(* Logix 5000 project; controller Sucrose_Main Emulate 5570 rev 20.12; software revision 20.01; part 18 of 30 *)
(* tags used below, declared in another part *)
   Alarm_ACK_Master_Timer : TIMER;
   DO_E22_6 : ALIAS FOR FLX_E22:6:O;   // Discrete Output EN2T_FLX 192.168.1.22
   DO_E22_7 : ALIAS FOR FLX_E22:7:O;   // Discrete Output EN2T_FLX 192.168.1.22
   FV740401_AOI : QSI_Flow_Valve;   // FV-74-04-01 SIP SUPPLY VALVE
   FV740501_AOI : QSI_Flow_Valve;   // FV-74-05-01 SIP SUPPLY TO PRE FILTER TRAIN 1 VALVE
   FV740502_AOI : QSI_Flow_Valve;   // FV-74-05-02 SIP SUPPLY TO FINAL FILTER TRAIN 1 VALVE
   FV740601_AOI : QSI_Flow_Valve;   // FV-74-06-01 SIP SUPPLY TO PRE FILTER TRAIN 2 VALVE
   FV740602_AOI : QSI_Flow_Valve;   // FV-74-06-02 SIP SUPPLY TO FINAL FILTER TRAIN 2 VALVE
   FV750501_AOI : QSI_Flow_Valve;   // FV-75-05-01 TRP-75-05-01 ISOLATION VALVE
   FV750502_AOI : QSI_Flow_Valve;   // FV-75-05-02 TRP-75-05-02 ISOLATION VALVE
   FV750503_AOI : QSI_Flow_Valve;   // FV-75-05-03 TRP-75-05-03 ISOLATION VALVE
   FV750504_AOI : QSI_Flow_Valve;   // FV-75-05-04 TRP-75-05-04 ISOLATION VALVE
   FV750601_AOI : QSI_Flow_Valve;   // FV-75-06-01 TRP-75-06-01 ISOLATION VALVE
   FV750602_AOI : QSI_Flow_Valve;   // FV-75-06-02 TRP-75-06-02 ISOLATION VALVE
   FV750603_AOI : QSI_Flow_Valve;   // FV-75-06-03 TRP-75-06-03 ISOLATION VALVE
   FV750604_AOI : QSI_Flow_Valve;   // FV-75-06-04 TRP-75-06-04 ISOLATION VALVE
   FV920501_AOI : QSI_Flow_Valve;   // FV-92-05-01 FLT-23-05-01 VENT VALVE
   FV930511_AOI : QSI_Flow_Valve;   // FV-93-05-11 PRE FILTER TRAIN 1 AIR BLOW OUTLET
   FV930512_AOI : QSI_Flow_Valve;   // FV-93-05-12 FINAL FILTER TRAIN 1 AIR BLOW OUTLET
   Sucrose_MM_Enable : BOOL;
   SucroseCIP_FILTRATION_REMOTE : CIP_REMOTE;
   SucroseFiltration : Area_Program;

PROGRAM FiltrationArea_EN2T_IO_Discrete_DO_E22_6   (* main routine MainRoutine *)

ROUTINE _00_FV740401   (* ladder *)
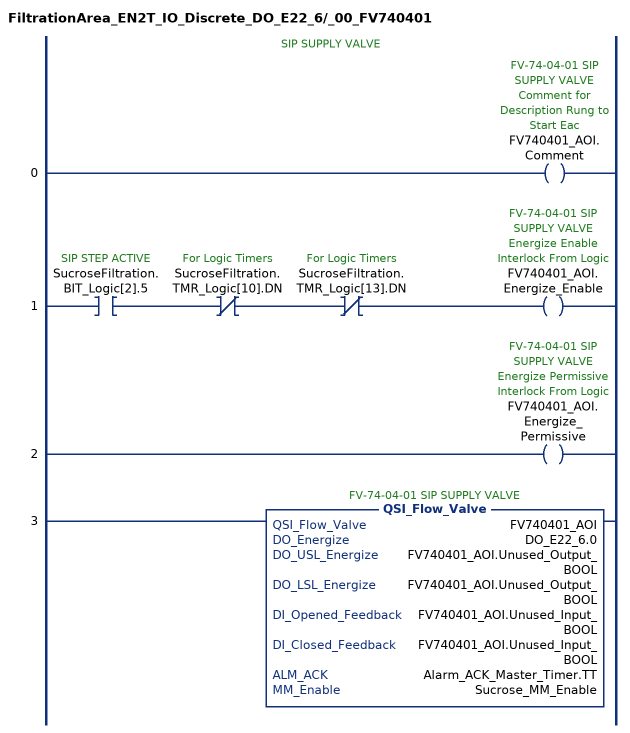
   // SIP SUPPLY VALVE
   0: OTE(FV740401_AOI.Comment);
   1: XIC(SucroseFiltration.BIT_Logic[2].5)XIO(SucroseFiltration.TMR_Logic[10].DN)XIO(SucroseFiltration.TMR_Logic[13].DN)OTE(FV740401_AOI.Energize_Enable);
   2: OTE(FV740401_AOI.Energize_Permissive);
   3: QSI_Flow_Valve(FV740401_AOI,DO_E22_6.0,FV740401_AOI.Unused_Output_BOOL,FV740401_AOI.Unused_Output_BOOL,FV740401_AOI.Unused_Input_BOOL,FV740401_AOI.Unused_Input_BOOL,Alarm_ACK_Master_Timer.TT,Sucrose_MM_Enable);
END_ROUTINE

ROUTINE _01_FV740501   (* ladder *)
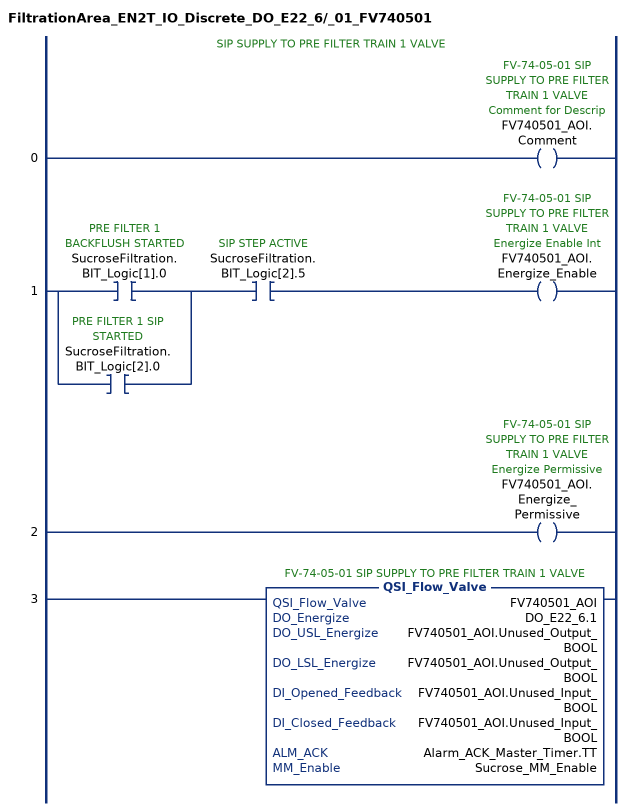
   // SIP SUPPLY TO PRE FILTER TRAIN 1 VALVE
   0: OTE(FV740501_AOI.Comment);
   1: [XIC(SucroseFiltration.BIT_Logic[1].0) ,XIC(SucroseFiltration.BIT_Logic[2].0) ]XIC(SucroseFiltration.BIT_Logic[2].5)OTE(FV740501_AOI.Energize_Enable);
   2: OTE(FV740501_AOI.Energize_Permissive);
   3: QSI_Flow_Valve(FV740501_AOI,DO_E22_6.1,FV740501_AOI.Unused_Output_BOOL,FV740501_AOI.Unused_Output_BOOL,FV740501_AOI.Unused_Input_BOOL,FV740501_AOI.Unused_Input_BOOL,Alarm_ACK_Master_Timer.TT,Sucrose_MM_Enable);
END_ROUTINE

ROUTINE _02_FV740502   (* ladder *)
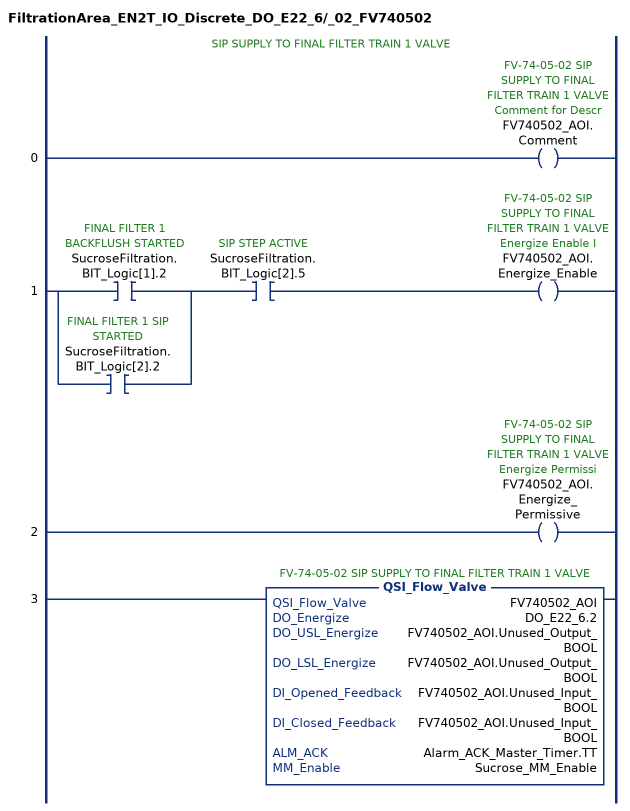
   // SIP SUPPLY TO FINAL FILTER TRAIN 1 VALVE
   0: OTE(FV740502_AOI.Comment);
   1: [XIC(SucroseFiltration.BIT_Logic[1].2) ,XIC(SucroseFiltration.BIT_Logic[2].2) ]XIC(SucroseFiltration.BIT_Logic[2].5)OTE(FV740502_AOI.Energize_Enable);
   2: OTE(FV740502_AOI.Energize_Permissive);
   3: QSI_Flow_Valve(FV740502_AOI,DO_E22_6.2,FV740502_AOI.Unused_Output_BOOL,FV740502_AOI.Unused_Output_BOOL,FV740502_AOI.Unused_Input_BOOL,FV740502_AOI.Unused_Input_BOOL,Alarm_ACK_Master_Timer.TT,Sucrose_MM_Enable);
END_ROUTINE

ROUTINE _03_FV740601   (* ladder *)
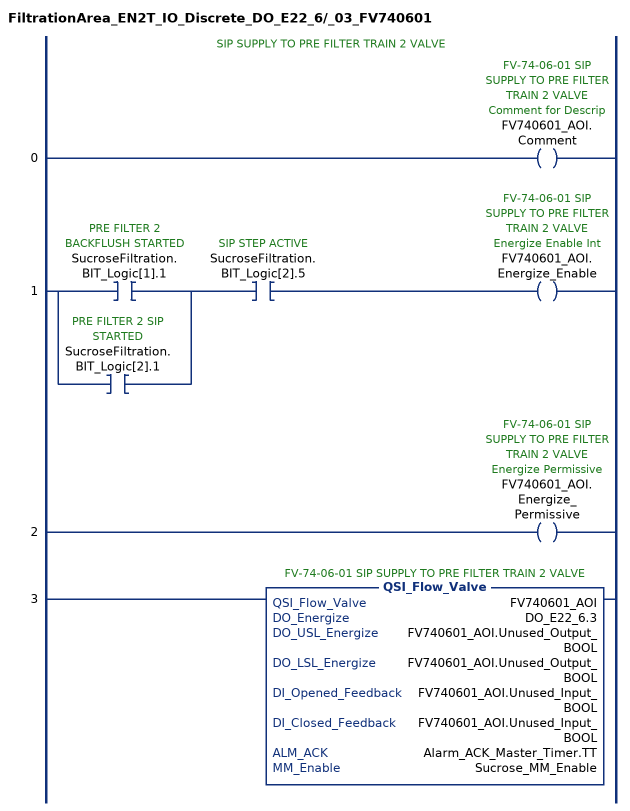
   // SIP SUPPLY TO PRE FILTER TRAIN 2 VALVE
   0: OTE(FV740601_AOI.Comment);
   1: [XIC(SucroseFiltration.BIT_Logic[1].1) ,XIC(SucroseFiltration.BIT_Logic[2].1) ]XIC(SucroseFiltration.BIT_Logic[2].5)OTE(FV740601_AOI.Energize_Enable);
   2: OTE(FV740601_AOI.Energize_Permissive);
   3: QSI_Flow_Valve(FV740601_AOI,DO_E22_6.3,FV740601_AOI.Unused_Output_BOOL,FV740601_AOI.Unused_Output_BOOL,FV740601_AOI.Unused_Input_BOOL,FV740601_AOI.Unused_Input_BOOL,Alarm_ACK_Master_Timer.TT,Sucrose_MM_Enable);
END_ROUTINE

ROUTINE _04_FV740602   (* ladder *)
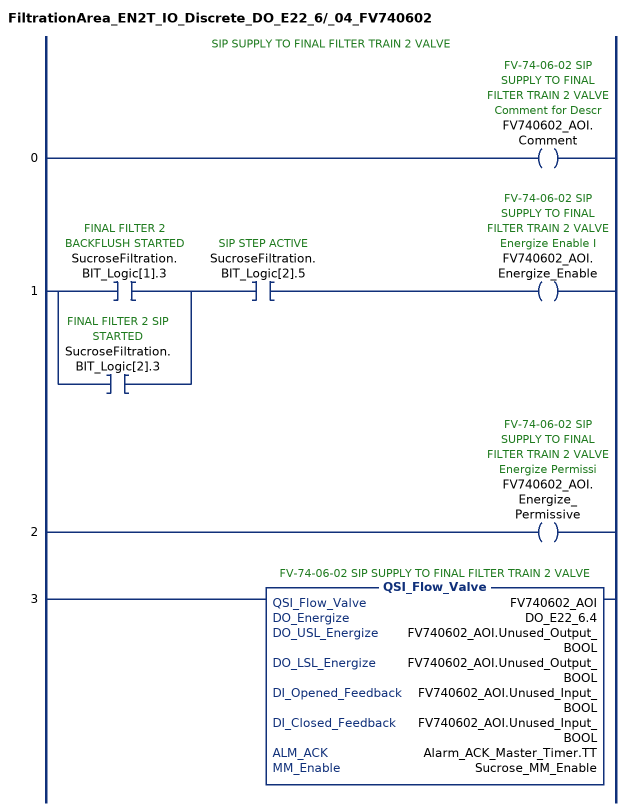
   // SIP SUPPLY TO FINAL FILTER TRAIN 2 VALVE
   0: OTE(FV740602_AOI.Comment);
   1: [XIC(SucroseFiltration.BIT_Logic[1].3) ,XIC(SucroseFiltration.BIT_Logic[2].3) ]XIC(SucroseFiltration.BIT_Logic[2].5)OTE(FV740602_AOI.Energize_Enable);
   2: OTE(FV740602_AOI.Energize_Permissive);
   3: QSI_Flow_Valve(FV740602_AOI,DO_E22_6.4,FV740602_AOI.Unused_Output_BOOL,FV740602_AOI.Unused_Output_BOOL,FV740602_AOI.Unused_Input_BOOL,FV740602_AOI.Unused_Input_BOOL,Alarm_ACK_Master_Timer.TT,Sucrose_MM_Enable);
END_ROUTINE

ROUTINE _05_FV750501   (* ladder *)
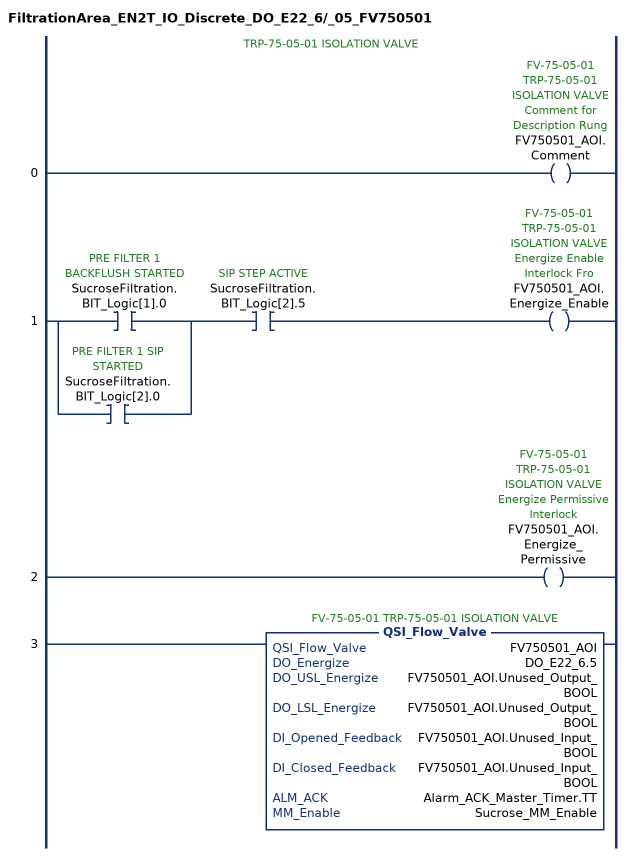
   // TRP-75-05-01 ISOLATION VALVE
   0: OTE(FV750501_AOI.Comment);
   1: [XIC(SucroseFiltration.BIT_Logic[1].0) ,XIC(SucroseFiltration.BIT_Logic[2].0) ]XIC(SucroseFiltration.BIT_Logic[2].5)OTE(FV750501_AOI.Energize_Enable);
   2: OTE(FV750501_AOI.Energize_Permissive);
   3: QSI_Flow_Valve(FV750501_AOI,DO_E22_6.5,FV750501_AOI.Unused_Output_BOOL,FV750501_AOI.Unused_Output_BOOL,FV750501_AOI.Unused_Input_BOOL,FV750501_AOI.Unused_Input_BOOL,Alarm_ACK_Master_Timer.TT,Sucrose_MM_Enable);
END_ROUTINE

ROUTINE _06_FV750502   (* ladder *)
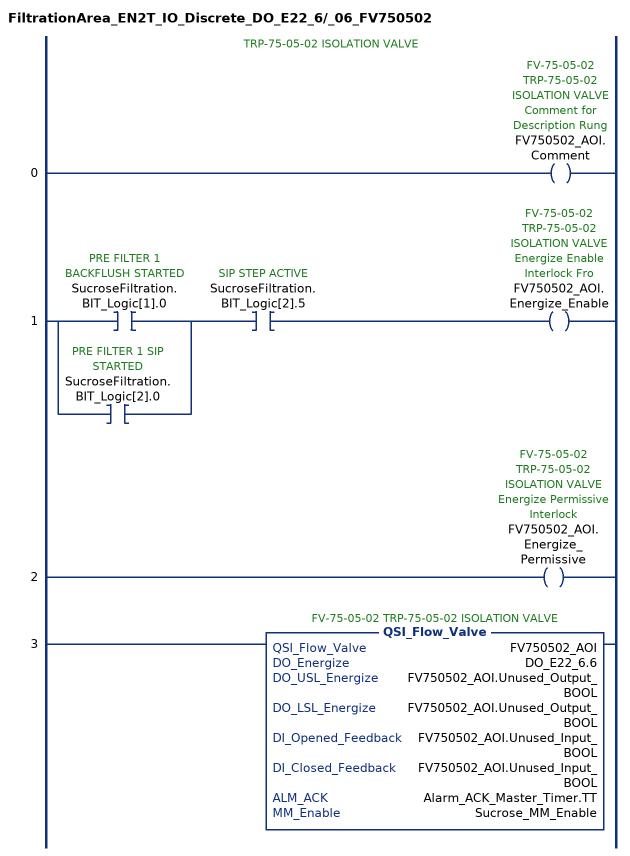
   // TRP-75-05-02 ISOLATION VALVE
   0: OTE(FV750502_AOI.Comment);
   1: [XIC(SucroseFiltration.BIT_Logic[1].0) ,XIC(SucroseFiltration.BIT_Logic[2].0) ]XIC(SucroseFiltration.BIT_Logic[2].5)OTE(FV750502_AOI.Energize_Enable);
   2: OTE(FV750502_AOI.Energize_Permissive);
   3: QSI_Flow_Valve(FV750502_AOI,DO_E22_6.6,FV750502_AOI.Unused_Output_BOOL,FV750502_AOI.Unused_Output_BOOL,FV750502_AOI.Unused_Input_BOOL,FV750502_AOI.Unused_Input_BOOL,Alarm_ACK_Master_Timer.TT,Sucrose_MM_Enable);
END_ROUTINE

ROUTINE _07_FV750503   (* ladder *)
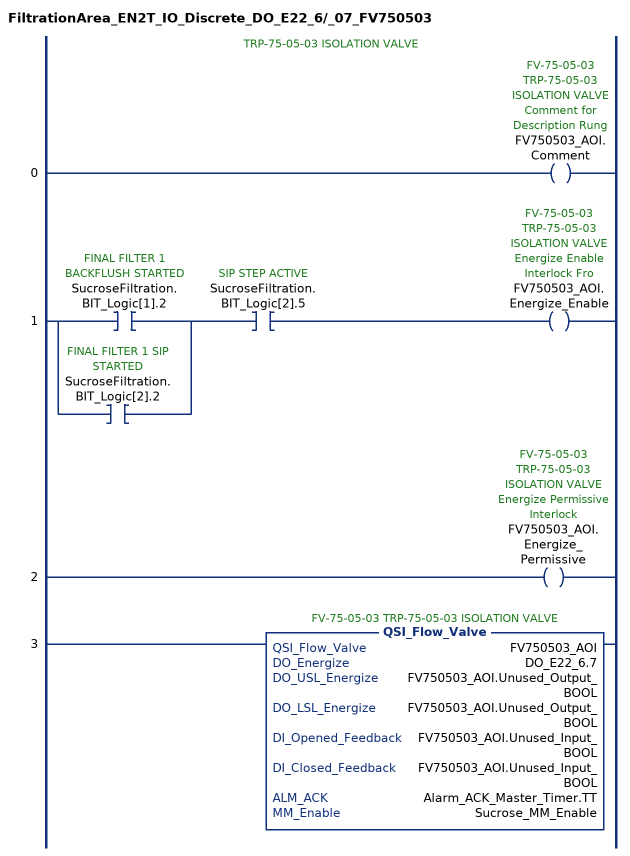
   // TRP-75-05-03 ISOLATION VALVE
   0: OTE(FV750503_AOI.Comment);
   1: [XIC(SucroseFiltration.BIT_Logic[1].2) ,XIC(SucroseFiltration.BIT_Logic[2].2) ]XIC(SucroseFiltration.BIT_Logic[2].5)OTE(FV750503_AOI.Energize_Enable);
   2: OTE(FV750503_AOI.Energize_Permissive);
   3: QSI_Flow_Valve(FV750503_AOI,DO_E22_6.7,FV750503_AOI.Unused_Output_BOOL,FV750503_AOI.Unused_Output_BOOL,FV750503_AOI.Unused_Input_BOOL,FV750503_AOI.Unused_Input_BOOL,Alarm_ACK_Master_Timer.TT,Sucrose_MM_Enable);
END_ROUTINE

ROUTINE _08_FV750504   (* ladder *)
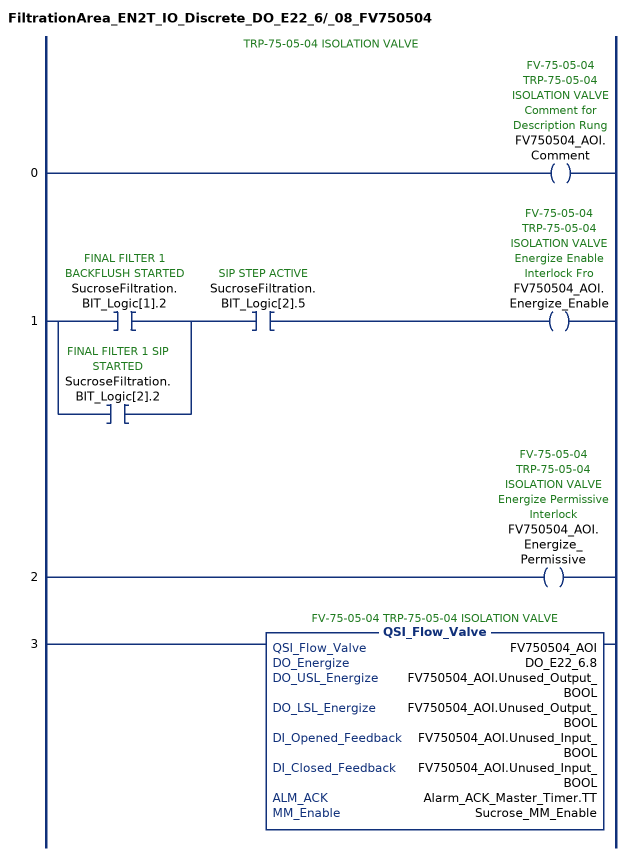
   // TRP-75-05-04 ISOLATION VALVE
   0: OTE(FV750504_AOI.Comment);
   1: [XIC(SucroseFiltration.BIT_Logic[1].2) ,XIC(SucroseFiltration.BIT_Logic[2].2) ]XIC(SucroseFiltration.BIT_Logic[2].5)OTE(FV750504_AOI.Energize_Enable);
   2: OTE(FV750504_AOI.Energize_Permissive);
   3: QSI_Flow_Valve(FV750504_AOI,DO_E22_6.8,FV750504_AOI.Unused_Output_BOOL,FV750504_AOI.Unused_Output_BOOL,FV750504_AOI.Unused_Input_BOOL,FV750504_AOI.Unused_Input_BOOL,Alarm_ACK_Master_Timer.TT,Sucrose_MM_Enable);
END_ROUTINE

ROUTINE _09_FV750601   (* ladder *)
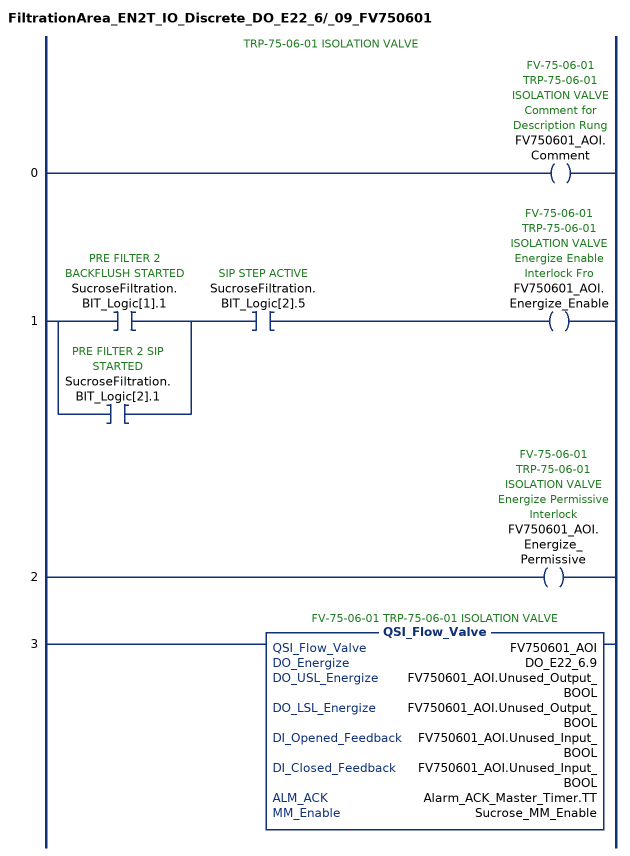
   // TRP-75-06-01 ISOLATION VALVE
   0: OTE(FV750601_AOI.Comment);
   1: [XIC(SucroseFiltration.BIT_Logic[1].1) ,XIC(SucroseFiltration.BIT_Logic[2].1) ]XIC(SucroseFiltration.BIT_Logic[2].5)OTE(FV750601_AOI.Energize_Enable);
   2: OTE(FV750601_AOI.Energize_Permissive);
   3: QSI_Flow_Valve(FV750601_AOI,DO_E22_6.9,FV750601_AOI.Unused_Output_BOOL,FV750601_AOI.Unused_Output_BOOL,FV750601_AOI.Unused_Input_BOOL,FV750601_AOI.Unused_Input_BOOL,Alarm_ACK_Master_Timer.TT,Sucrose_MM_Enable);
END_ROUTINE

ROUTINE _10_FV750602   (* ladder *)
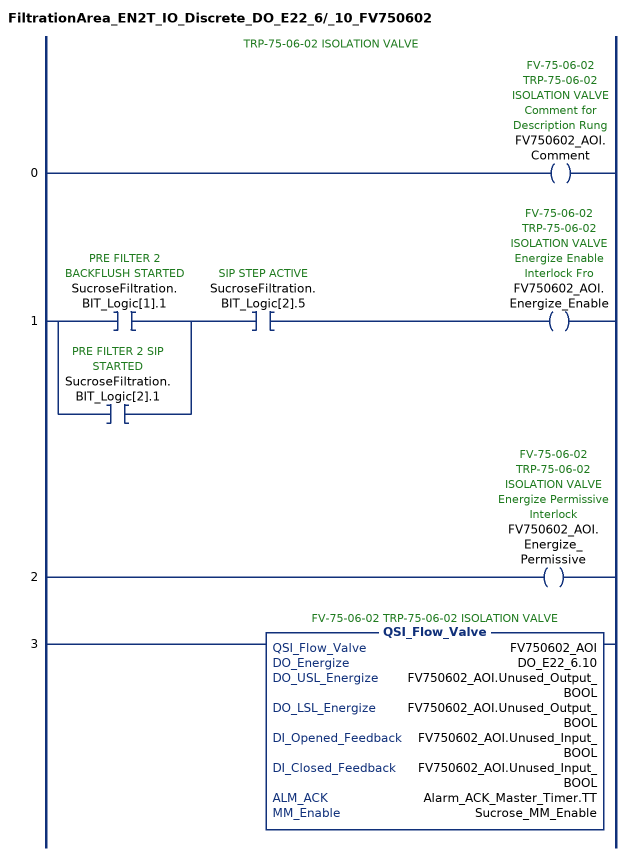
   // TRP-75-06-02 ISOLATION VALVE
   0: OTE(FV750602_AOI.Comment);
   1: [XIC(SucroseFiltration.BIT_Logic[1].1) ,XIC(SucroseFiltration.BIT_Logic[2].1) ]XIC(SucroseFiltration.BIT_Logic[2].5)OTE(FV750602_AOI.Energize_Enable);
   2: OTE(FV750602_AOI.Energize_Permissive);
   3: QSI_Flow_Valve(FV750602_AOI,DO_E22_6.10,FV750602_AOI.Unused_Output_BOOL,FV750602_AOI.Unused_Output_BOOL,FV750602_AOI.Unused_Input_BOOL,FV750602_AOI.Unused_Input_BOOL,Alarm_ACK_Master_Timer.TT,Sucrose_MM_Enable);
END_ROUTINE

ROUTINE _11_FV750603   (* ladder *)
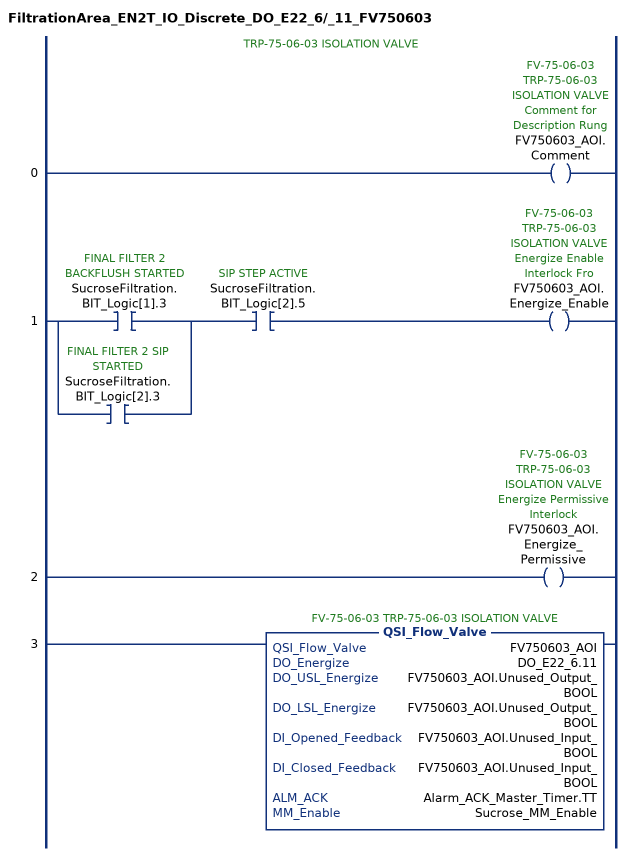
   // TRP-75-06-03 ISOLATION VALVE
   0: OTE(FV750603_AOI.Comment);
   1: [XIC(SucroseFiltration.BIT_Logic[1].3) ,XIC(SucroseFiltration.BIT_Logic[2].3) ]XIC(SucroseFiltration.BIT_Logic[2].5)OTE(FV750603_AOI.Energize_Enable);
   2: OTE(FV750603_AOI.Energize_Permissive);
   3: QSI_Flow_Valve(FV750603_AOI,DO_E22_6.11,FV750603_AOI.Unused_Output_BOOL,FV750603_AOI.Unused_Output_BOOL,FV750603_AOI.Unused_Input_BOOL,FV750603_AOI.Unused_Input_BOOL,Alarm_ACK_Master_Timer.TT,Sucrose_MM_Enable);
END_ROUTINE

ROUTINE _12_FV930511   (* ladder *)
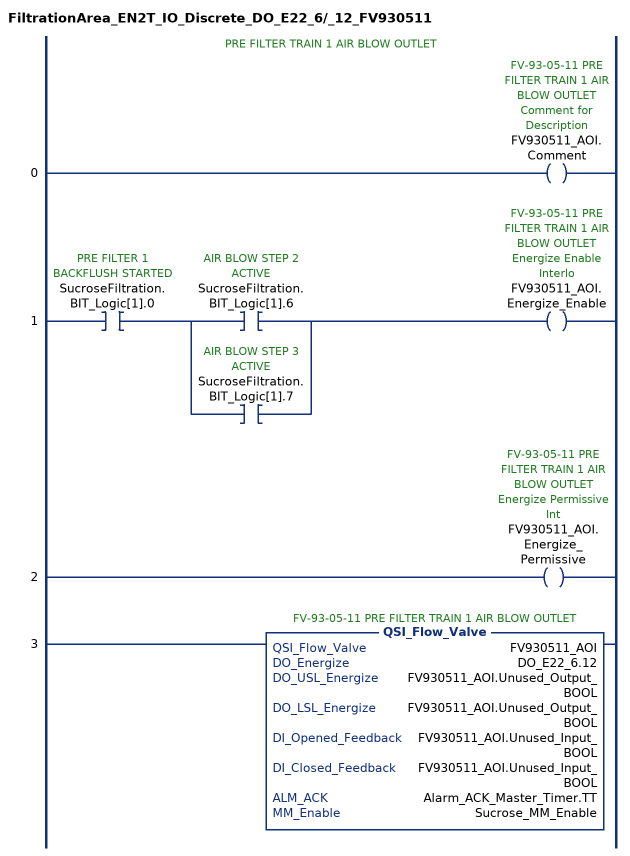
   // PRE FILTER TRAIN 1 AIR BLOW OUTLET
   0: OTE(FV930511_AOI.Comment);
   1: XIC(SucroseFiltration.BIT_Logic[1].0)[XIC(SucroseFiltration.BIT_Logic[1].6) ,XIC(SucroseFiltration.BIT_Logic[1].7) ]OTE(FV930511_AOI.Energize_Enable);
   2: OTE(FV930511_AOI.Energize_Permissive);
   3: QSI_Flow_Valve(FV930511_AOI,DO_E22_6.12,FV930511_AOI.Unused_Output_BOOL,FV930511_AOI.Unused_Output_BOOL,FV930511_AOI.Unused_Input_BOOL,FV930511_AOI.Unused_Input_BOOL,Alarm_ACK_Master_Timer.TT,Sucrose_MM_Enable);
END_ROUTINE

ROUTINE _13_FV930512   (* ladder *)
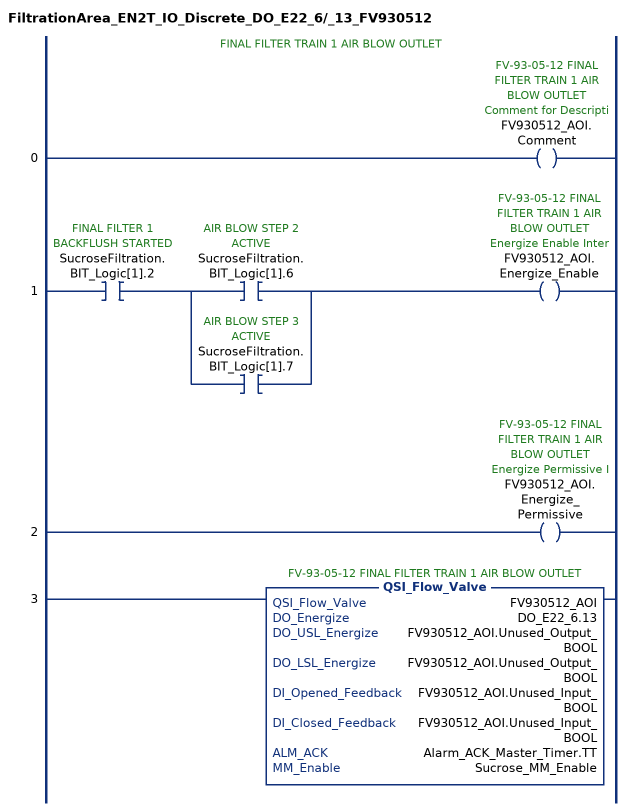
   // FINAL FILTER TRAIN 1 AIR BLOW OUTLET
   0: OTE(FV930512_AOI.Comment);
   1: XIC(SucroseFiltration.BIT_Logic[1].2)[XIC(SucroseFiltration.BIT_Logic[1].6) ,XIC(SucroseFiltration.BIT_Logic[1].7) ]OTE(FV930512_AOI.Energize_Enable);
   2: OTE(FV930512_AOI.Energize_Permissive);
   3: QSI_Flow_Valve(FV930512_AOI,DO_E22_6.13,FV930512_AOI.Unused_Output_BOOL,FV930512_AOI.Unused_Output_BOOL,FV930512_AOI.Unused_Input_BOOL,FV930512_AOI.Unused_Input_BOOL,Alarm_ACK_Master_Timer.TT,Sucrose_MM_Enable);
END_ROUTINE

ROUTINE MainRoutine   (* ladder *)
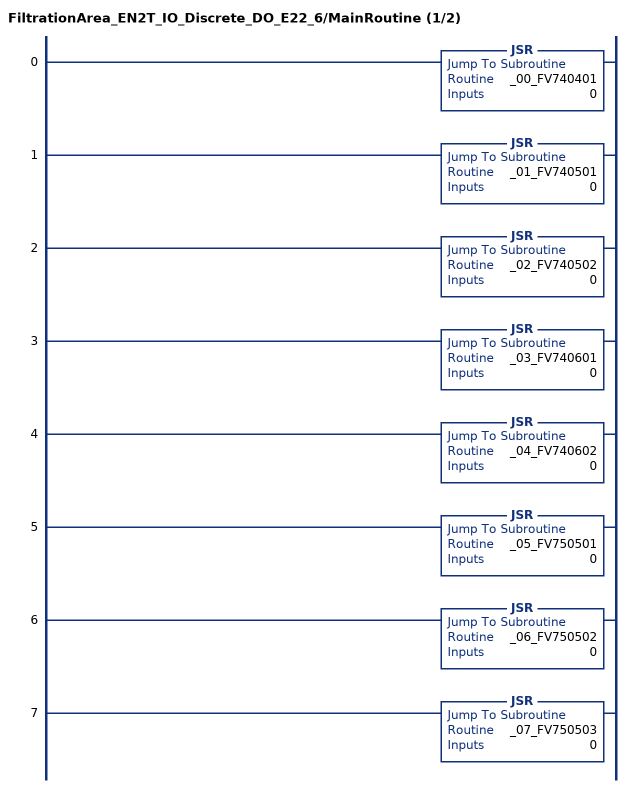
   0: JSR(_00_FV740401,0);
   1: JSR(_01_FV740501,0);
   2: JSR(_02_FV740502,0);
   3: JSR(_03_FV740601,0);
   4: JSR(_04_FV740602,0);
   5: JSR(_05_FV750501,0);
   6: JSR(_06_FV750502,0);
   7: JSR(_07_FV750503,0);
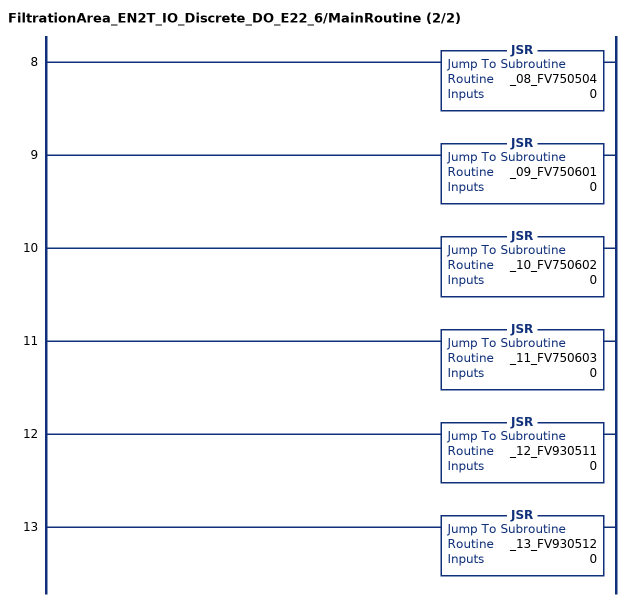
   8: JSR(_08_FV750504,0);
   9: JSR(_09_FV750601,0);
   10: JSR(_10_FV750602,0);
   11: JSR(_11_FV750603,0);
   12: JSR(_12_FV930511,0);
   13: JSR(_13_FV930512,0);
END_ROUTINE
END_PROGRAM

PROGRAM FiltrationArea_EN2T_IO_Discrete_DO_E22_7   (* main routine MainRoutine *)

ROUTINE _00_FV750604   (* ladder *)
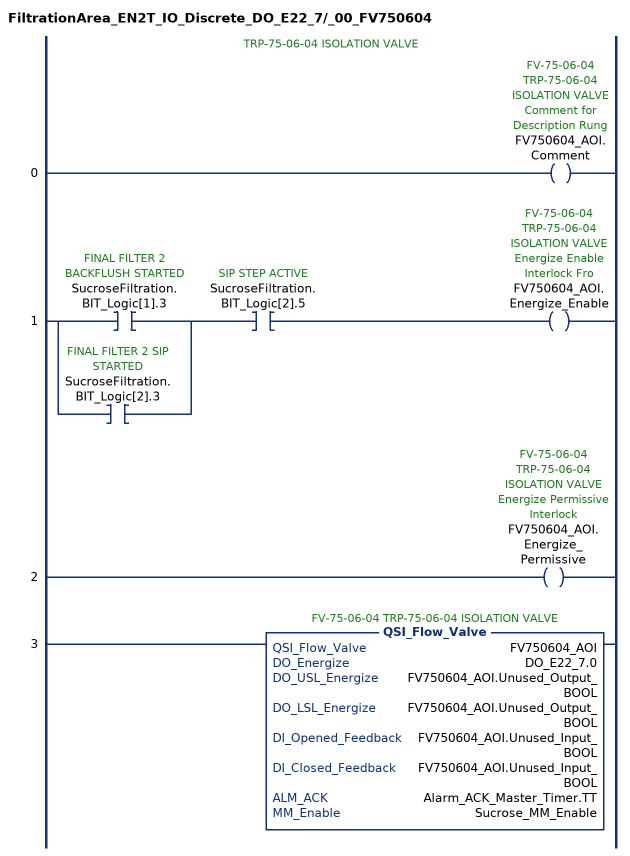
   // TRP-75-06-04 ISOLATION VALVE
   0: OTE(FV750604_AOI.Comment);
   1: [XIC(SucroseFiltration.BIT_Logic[1].3) ,XIC(SucroseFiltration.BIT_Logic[2].3) ]XIC(SucroseFiltration.BIT_Logic[2].5)OTE(FV750604_AOI.Energize_Enable);
   2: OTE(FV750604_AOI.Energize_Permissive);
   3: QSI_Flow_Valve(FV750604_AOI,DO_E22_7.0,FV750604_AOI.Unused_Output_BOOL,FV750604_AOI.Unused_Output_BOOL,FV750604_AOI.Unused_Input_BOOL,FV750604_AOI.Unused_Input_BOOL,Alarm_ACK_Master_Timer.TT,Sucrose_MM_Enable);
END_ROUTINE

ROUTINE _01_FV920501   (* ladder *)
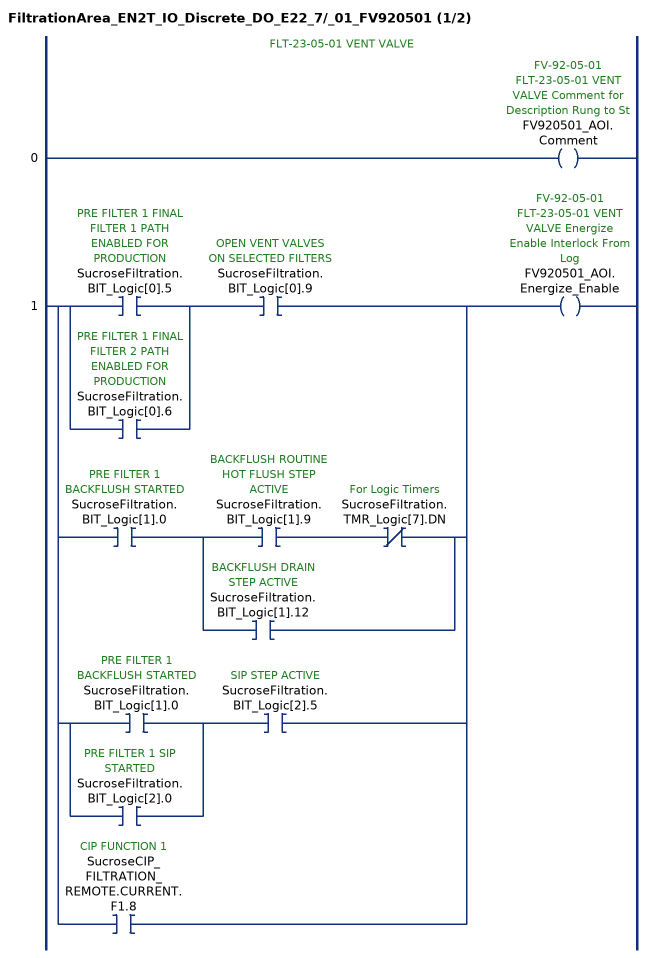
   // FLT-23-05-01 VENT VALVE
   0: OTE(FV920501_AOI.Comment);
   1: [[XIC(SucroseFiltration.BIT_Logic[0].5) ,XIC(SucroseFiltration.BIT_Logic[0].6) ] XIC(SucroseFiltration.BIT_Logic[0].9) ,XIC(SucroseFiltration.BIT_Logic[1].0) [XIC(SucroseFiltration.BIT_Logic[1].9) XIO(SucroseFiltration.TMR_Logic[7].DN) ,XIC(SucroseFiltration.BIT_Logic[1].12) ] ,[XIC(SucroseFiltration.BIT_Logic[1].0) ,XIC(SucroseFiltration.BIT_Logic[2].0) ] XIC(SucroseFiltration.BIT_Logic[2].5) ,XIC(SucroseCIP_FILTRATION_REMOTE.CURRENT.F1.8) ]OTE(FV920501_AOI.Energize_Enable);
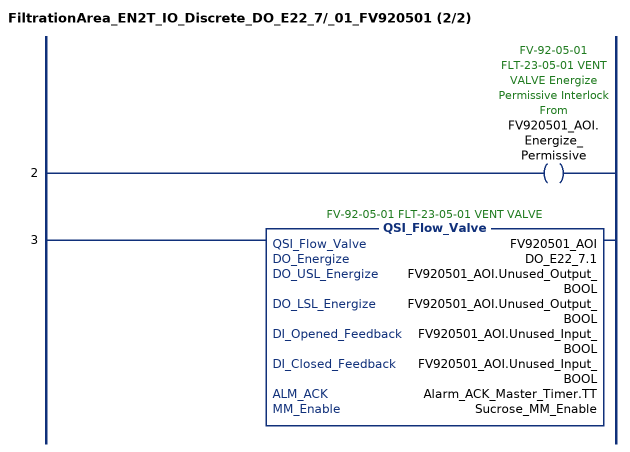
   2: OTE(FV920501_AOI.Energize_Permissive);
   3: QSI_Flow_Valve(FV920501_AOI,DO_E22_7.1,FV920501_AOI.Unused_Output_BOOL,FV920501_AOI.Unused_Output_BOOL,FV920501_AOI.Unused_Input_BOOL,FV920501_AOI.Unused_Input_BOOL,Alarm_ACK_Master_Timer.TT,Sucrose_MM_Enable);
END_ROUTINE
